Staubli VAL3: releaseObject.pgx

program releaseObject(num x_nIndex (dimensions=1))
begin
  switch nLinkedTo[x_nIndex]
    case 0
      call cnv0:releaseObject(nPosInQueue[x_nIndex])
    break
    case 1
      call cnv1:releaseObject(nPosInQueue[x_nIndex])
    break
  endSwitch
  nLinkedTo[x_nIndex]=-1
  nPosInQueue[x_nIndex]=-1
end
